// Mitsubishi GX Works2 project: PID_slave_test_fx3u_demo   PLC: FX3U/FX3UC

// global labels: Global1
VAR_GLOBAL
  Input_ManualMode AT M500 : BOOL;  (* Valg av Manuell "1" eller Auto "0" *)
  Input_OperationModus AT M501 : BOOL;  (* Valg av direkte "1" eller Revers "0" Regulering *)
  Input_IntegratorModus AT M502 : BOOL;  (* Valg av Integrator virkning på regulator *)
  Input_DerivatorModus AT M503 : BOOL;  (* Valg av Derivator virkning på regulator *)
  Input_SamplingsTime AT D200 : INT;  (* Samplingstid sendt til PID *)
  Output_PID AT D202 : REAL;  (* Utgangs signal sendt ut fra PID *)
  Input_Referance AT D204 : REAL;  (* Referanse verdi sendt til PID *)
  Input_Process AT D206 : REAL;  (* Prosess verdi Sendt til PID *)
  Input_ManualValue AT D208 : REAL;  (* Manuell verdi sendt til PID *)
  Input_NomValue AT D210 : REAL;  (* Nominelt pådrag *)
  Input_MaxPådrag AT D212 : REAL;  (* Max pådrag *)
  Input_MinPådrag AT D214 : REAL;  (* Min pådrag *)
  Input_Skalert_Samplingstid AT D216 : ARRAY [0..1] OF INT;  (* Samplingstid skalert til timer *)
  Input_KpValue AT D218 : REAL;  (* Valg av Kp verdi *)
  Input_TiValue AT D220 : REAL;  (* Valge av Ti verdi *)
  Input_TdValue AT D222 : REAL;  (* Valg av Td verdi *)
  Input_NValue AT D224 : REAL;  (* Valg av N verdi *)
  Input_TtValue AT D226 : REAL;  (* Valg av Tt verdi *)
  Input_FF_TtValue AT D228 : REAL;  (* Valg av Tt verdi til LeadLag blokk *)
  Input_FF_TnValue AT D230 : REAL;  (* Valg av Tn verdi til LeadLag blokk *)
  Input_FF_KLLValue AT D232 : REAL;  (* Valg av KLL verdi til LeadLag blokk *)
  Output_Leadlag AT D234 : REAL;  (* Utgangsignal sendt ut fra LeadLag blokk *)
  Output_Total AT D236 : REAL;  (* Totalt utgangsignal summert *)
  Input_ErrorValue AT D238 : REAL;  (* Beregnet avvik *)
  Input_AI_Raw AT D400 : INT;
  Output_AO_Raw AT D402 : INT;
  Storage_havardsinlillepikk AT D500 : INT;  (* Mellomlagrin av referanse verdi før omgjøring til flyttall *)
  anaDig AT D8260 : INT;
  digAna AT D8262 : INT;
  Storage_Filter_Output AT D502 : INT;  (* Utgangsverdi fra filter *)
  Tank_high AT M504 : BOOL;
  Tank_low AT M505 : BOOL;
  Tank_high_high AT M506 : BOOL;
  Tank_low_low AT M507 : BOOL;
  Tank_criticalHigh AT M508 : BOOL;
  Tank_criticalLow AT M509 : BOOL;
  Tank_normalHigh AT M510 : BOOL;
  Tank_normalLow AT M511 : BOOL;
  Acknowledge_normalHigh AT M512 : BOOL;
  Acknowledge_normalLow AT M513 : BOOL;
  Acknowledge_criticalHigh AT M514 : BOOL;
  Acknowledge_criticalLow AT M515 : BOOL;
  Pump AT Y012 : BOOL;
  Normal_ErrorSignal AT M516 : BOOL;
  Critical_ErrorSignal AT M517 : BOOL;
  Normal_ErrorCheck AT M518 : ARRAY [0..2] OF BOOL;
  Critical_ErrorCheck AT M519 : ARRAY [0..2] OF BOOL;
  Process_memory AT M520 : BOOL;
  Process AT M21 : BOOL;
  Power_failure AT M522 : BOOL;
  Acknowledge_powerFailure AT M523 : BOOL;
  Alarm_Lamp AT Y001 : BOOL;
  Communication_trouble AT X001 : BOOL;
  Communication_troubleRST AT Y002 : BOOL;
  Communication_troubleRSTCommand AT X021 : BOOL;
  Communication_rstFlag AT M1 : BOOL;
  Profibus_code AT D1000 : INT;
END_VAR

// task Task_01 (event TRUE, interval 0, priority 31): POU_01

PROGRAM POU_01
VAR
  My_PID_1 : My_PID;
  LeadLag_1 : LeadLag;
  Output_Adder_1 : Output_Adder;
  Filter_Midling_1 : Filter_Midling;
END_VAR
(* structured ladder/FBD written out as ST: instructions are called as NAME(EN, inputs, outputs); _pN, _eN, _tN stand for wires *)
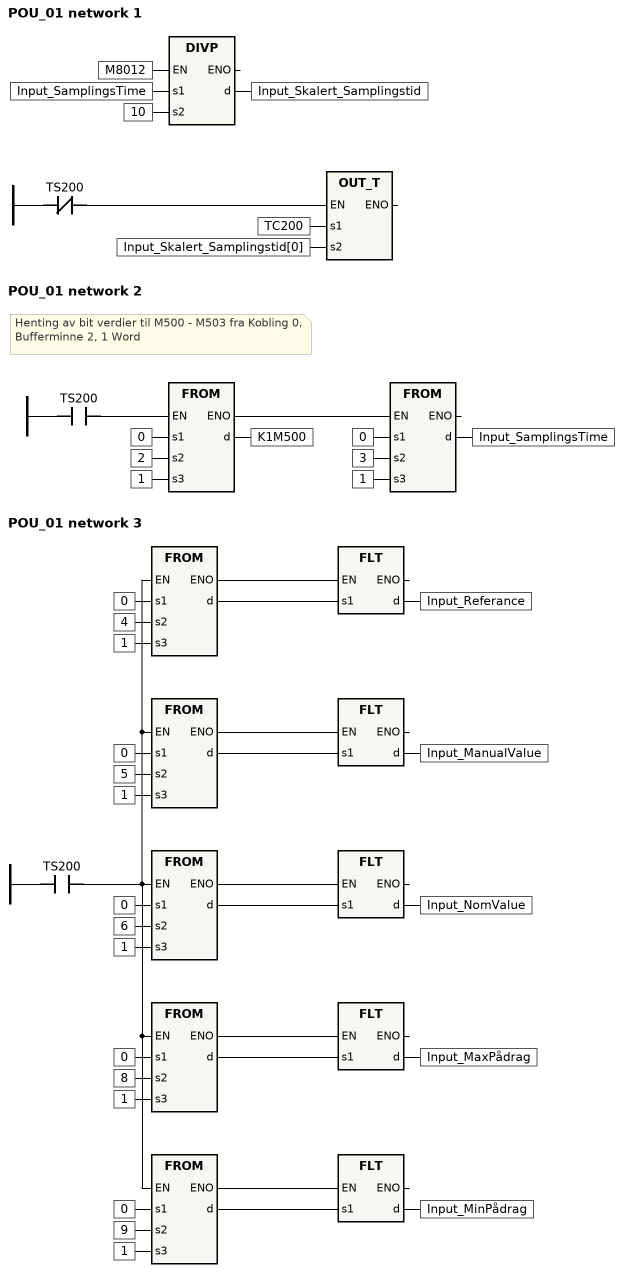
(* network 1 *)
DIVP(M8012, Input_SamplingsTime, 10, Input_Skalert_Samplingstid);
OUT_T(NOT TS200, TC200, Input_Skalert_Samplingstid[0]);
(* network 2 *)
(* Henting av bit verdier til M500 - M503 fra Kobling 0, Bufferminne 2, 1 Word *)
_e1 := FROM(TS200, 0, 2, 1, K1M500);
FROM(_e1, 0, 3, 1, Input_SamplingsTime);
(* network 3 *)
_e2 := FROM(TS200, 0, 4, 1, _t1);
FLT(_e2, _t1, Input_Referance);
_e4 := FROM(TS200, 0, 5, 1, _t3);
FLT(_e4, _t3, Input_ManualValue);
_e6 := FROM(TS200, 0, 6, 1, _t5);
FLT(_e6, _t5, Input_NomValue);
_e8 := FROM(TS200, 0, 8, 1, _t7);
FLT(_e8, _t7, Input_MaxPådrag);
_e10 := FROM(TS200, 0, 9, 1, _t9);
FLT(_e10, _t9, Input_MinPådrag);
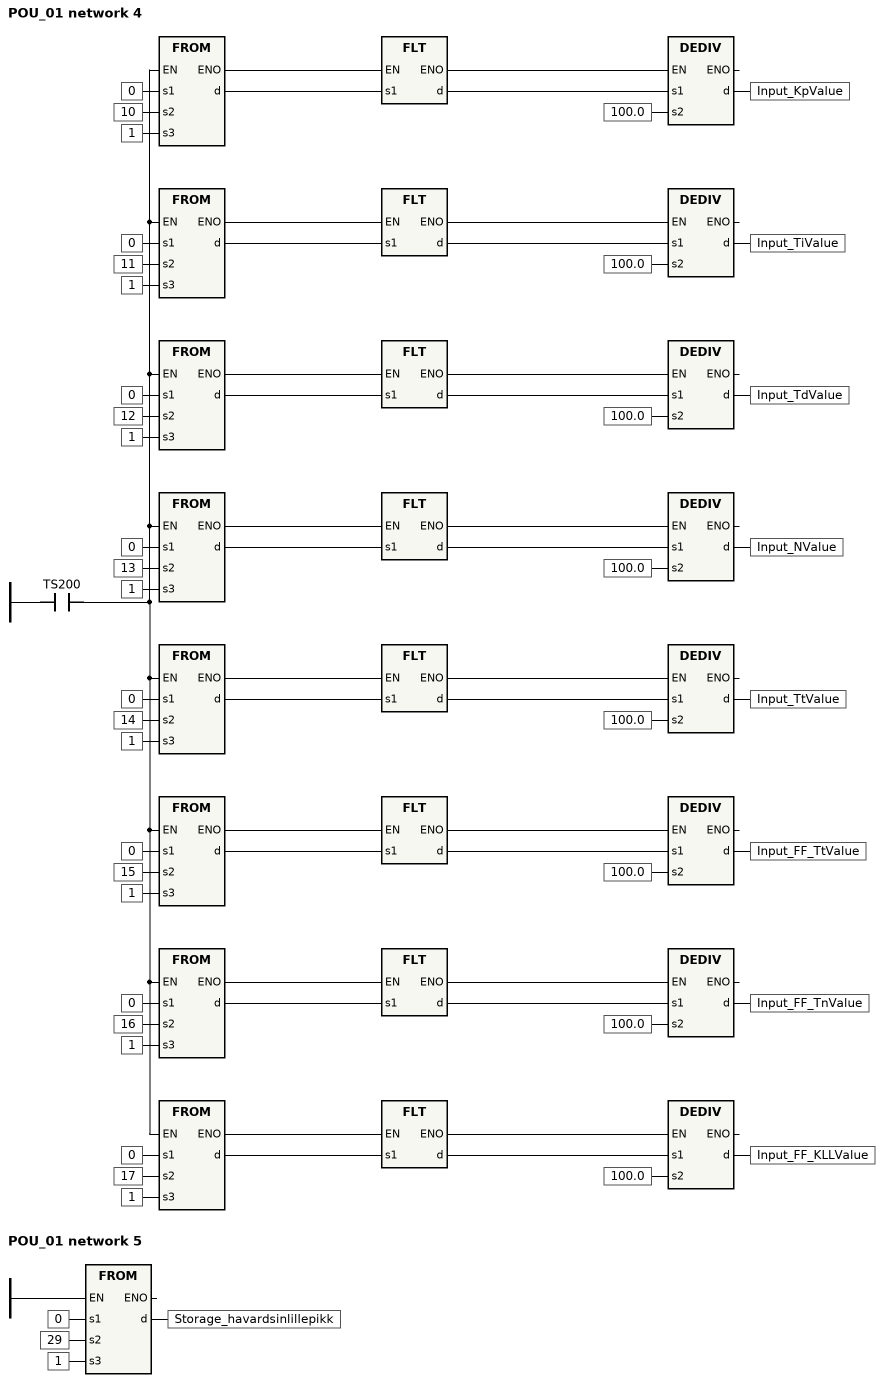
(* network 4 *)
_e2 := FROM(TS200, 0, 10, 1, _t1);
_e4 := FLT(_e2, _t1, _t3);
DEDIV(_e4, _t3, 100.0, Input_KpValue);
_e6 := FROM(TS200, 0, 11, 1, _t5);
_e8 := FLT(_e6, _t5, _t7);
DEDIV(_e8, _t7, 100.0, Input_TiValue);
_e10 := FROM(TS200, 0, 12, 1, _t9);
_e12 := FLT(_e10, _t9, _t11);
DEDIV(_e12, _t11, 100.0, Input_TdValue);
_e14 := FROM(TS200, 0, 13, 1, _t13);
_e16 := FLT(_e14, _t13, _t15);
DEDIV(_e16, _t15, 100.0, Input_NValue);
_e18 := FROM(TS200, 0, 14, 1, _t17);
_e20 := FLT(_e18, _t17, _t19);
DEDIV(_e20, _t19, 100.0, Input_TtValue);
_e22 := FROM(TS200, 0, 15, 1, _t21);
_e24 := FLT(_e22, _t21, _t23);
DEDIV(_e24, _t23, 100.0, Input_FF_TtValue);
_e26 := FROM(TS200, 0, 16, 1, _t25);
_e28 := FLT(_e26, _t25, _t27);
DEDIV(_e28, _t27, 100.0, Input_FF_TnValue);
_e30 := FROM(TS200, 0, 17, 1, _t29);
_e32 := FLT(_e30, _t29, _t31);
DEDIV(_e32, _t31, 100.0, Input_FF_KLLValue);
(* network 5 *)
FROM(TRUE, 0, 29, 1, Storage_havardsinlillepikk);
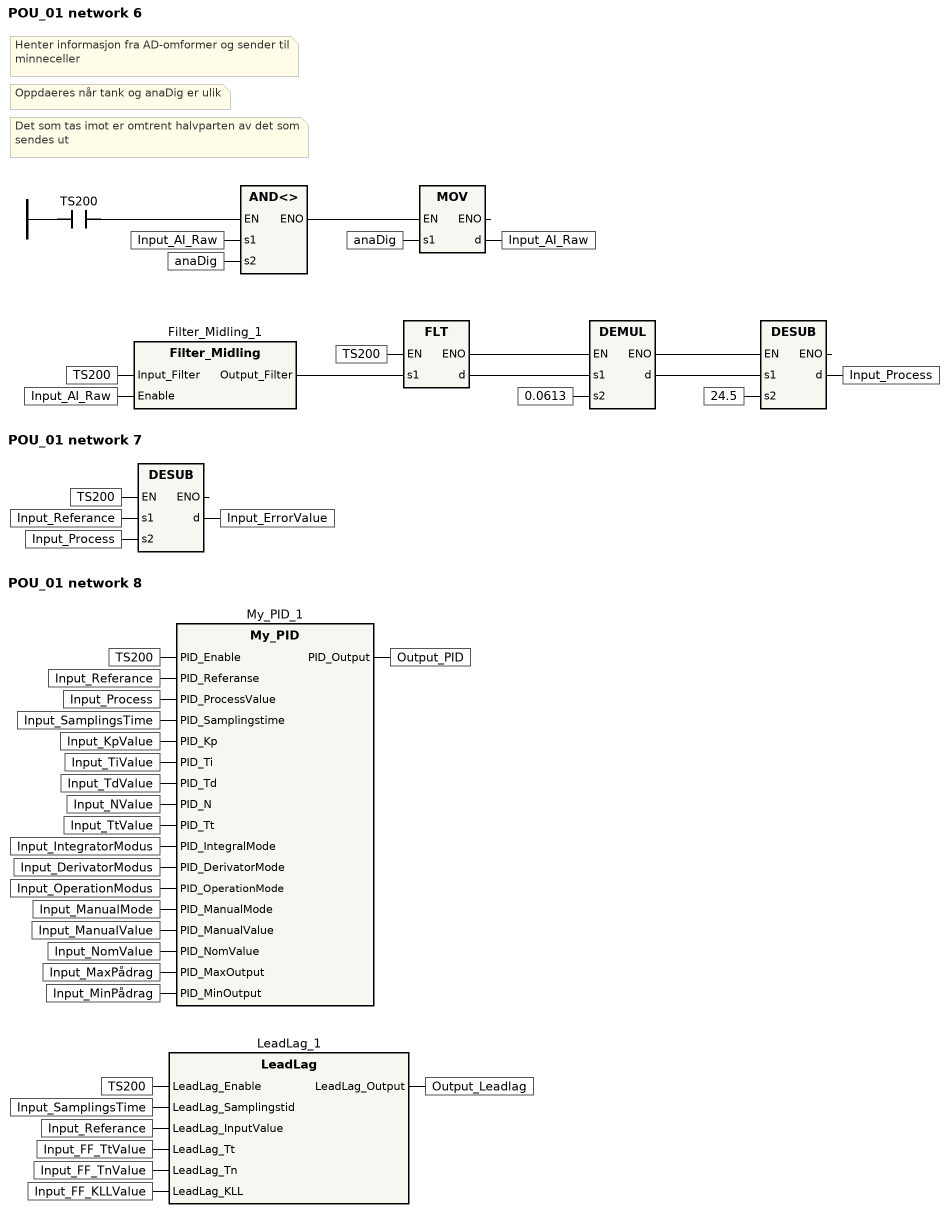
(* network 6 *)
(* Henter informasjon fra AD-omformer og sender til minneceller *)
(* Oppdaeres når tank og anaDig er ulik *)
(* Det som tas imot er omtrent halvparten av det som sendes ut *)
_e1 := AND<>(TS200, Input_AI_Raw, anaDig);
MOV(_e1, anaDig, Input_AI_Raw);
Filter_Midling_1(Input_Filter := TS200, Enable := Input_AI_Raw);
_e3 := FLT(TS200, Filter_Midling_1.Output_Filter, _t2);
_e5 := DEMUL(_e3, _t2, 0.0613, _t4);
DESUB(_e5, _t4, 24.5, Input_Process);
(* network 7 *)
DESUB(TS200, Input_Referance, Input_Process, Input_ErrorValue);
(* network 8 *)
My_PID_1(PID_Enable := TS200, PID_Referanse := Input_Referance, PID_ProcessValue := Input_Process, PID_Samplingstime := Input_SamplingsTime, PID_Kp := Input_KpValue, PID_Ti := Input_TiValue, PID_Td := Input_TdValue, PID_N := Input_NValue, PID_Tt := Input_TtValue, PID_IntegralMode := Input_IntegratorModus, PID_DerivatorMode := Input_DerivatorModus, PID_OperationMode := Input_OperationModus, PID_ManualMode := Input_ManualMode, PID_ManualValue := Input_ManualValue, PID_NomValue := Input_NomValue, PID_MaxOutput := Input_MaxPådrag, PID_MinOutput := Input_MinPådrag, PID_Output => Output_PID);
LeadLag_1(LeadLag_Enable := TS200, LeadLag_Samplingstid := Input_SamplingsTime, LeadLag_InputValue := Input_Referance, LeadLag_Tt := Input_FF_TtValue, LeadLag_Tn := Input_FF_TnValue, LeadLag_KLL := Input_FF_KLLValue, LeadLag_Output => Output_Leadlag);
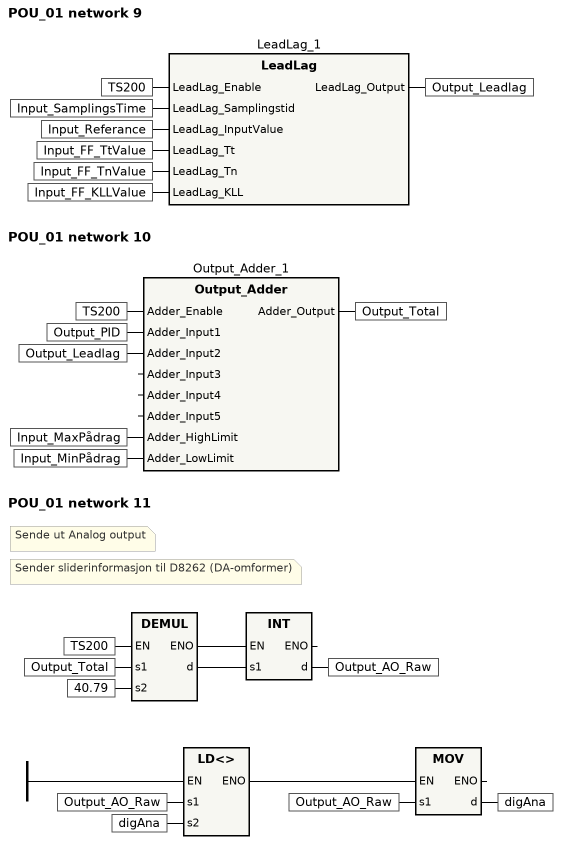
(* network 9 *)
LeadLag_1(LeadLag_Enable := TS200, LeadLag_Samplingstid := Input_SamplingsTime, LeadLag_InputValue := Input_Referance, LeadLag_Tt := Input_FF_TtValue, LeadLag_Tn := Input_FF_TnValue, LeadLag_KLL := Input_FF_KLLValue, LeadLag_Output => Output_Leadlag);
(* network 10 *)
Output_Adder_1(Adder_Enable := TS200, Adder_Input1 := Output_PID, Adder_Input2 := Output_Leadlag, Adder_HighLimit := Input_MaxPådrag, Adder_LowLimit := Input_MinPådrag, Adder_Output => Output_Total);
(* network 11 *)
(* Sende ut Analog output *)
(* Sender sliderinformasjon til D8262 (DA-omformer) *)
_e2 := DEMUL(TS200, Output_Total, 40.79, _t1);
INT(_e2, _t1, Output_AO_Raw);
_e3 := LD<>(TRUE, Output_AO_Raw, digAna);
MOV(_e3, Output_AO_Raw, digAna);
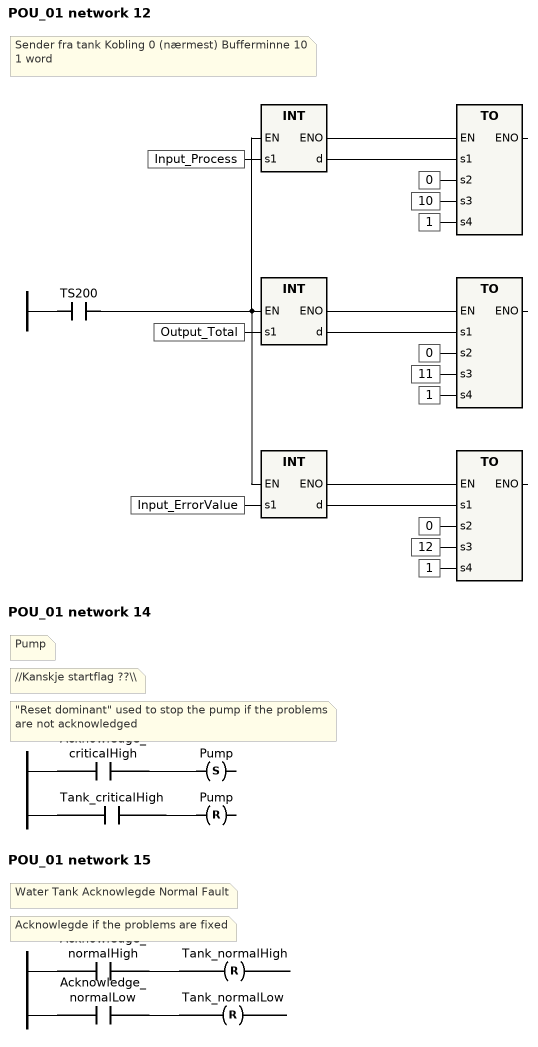
(* network 12 *)
(* Sender fra tank Kobling 0 (nærmest) Bufferminne 10           1 word *)
_e2 := INT(TS200, Input_Process, _t1);
TO(_e2, _t1, 0, 10, 1);
_e4 := INT(TS200, Output_Total, _t3);
TO(_e4, _t3, 0, 11, 1);
_e6 := INT(TS200, Input_ErrorValue, _t5);
TO(_e6, _t5, 0, 12, 1);
(* network 14 *)
(* Pump *)
(* //Kanskje startflag ??\\ *)
(* "Reset dominant" used to stop the pump if the problems are not acknowledged *)
SET(Acknowledge_criticalHigh, Pump);
RST(Tank_criticalHigh, Pump);
(* network 15 *)
(* Water Tank Acknowlegde Normal Fault *)
(* Acknowlegde if the problems are fixed *)
RST(Acknowledge_normalHigh, Tank_normalHigh);
RST(Acknowledge_normalLow, Tank_normalLow);
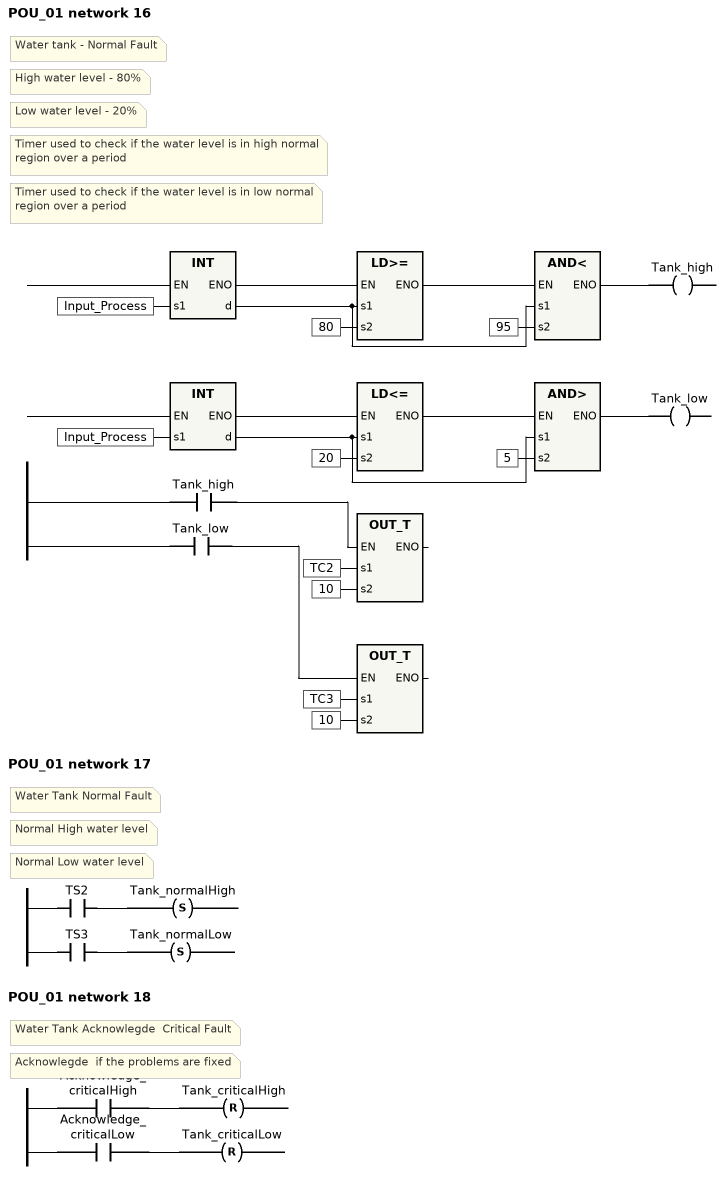
(* network 16 *)
(* Water tank - Normal Fault *)
(* High water level - 80% *)
(* Low water level - 20% *)
(* Timer used to check if the water level is in high normal region over a period *)
(* Timer used to check if the water level is in low normal region over a period *)
_e2 := INT(TRUE, Input_Process, _t1);
_e3 := LD>=(_e2, _t1, 80);
_e4 := AND<(_e3, _t1, 95);
Tank_high := _e4;
_e6 := INT(TRUE, Input_Process, _t5);
_e7 := LD<=(_e6, _t5, 20);
_e8 := AND>(_e7, _t5, 5);
Tank_low := _e8;
OUT_T(Tank_high, TC2, 10);
OUT_T(Tank_low, TC3, 10);
(* network 17 *)
(* Water Tank Normal Fault *)
(* Normal High water level *)
(* Normal Low water level *)
SET(TS2, Tank_normalHigh);
SET(TS3, Tank_normalLow);
(* network 18 *)
(* Water Tank Acknowlegde  Critical Fault *)
(* Acknowlegde  if the problems are fixed *)
RST(Acknowledge_criticalHigh, Tank_criticalHigh);
RST(Acknowledge_criticalLow, Tank_criticalLow);
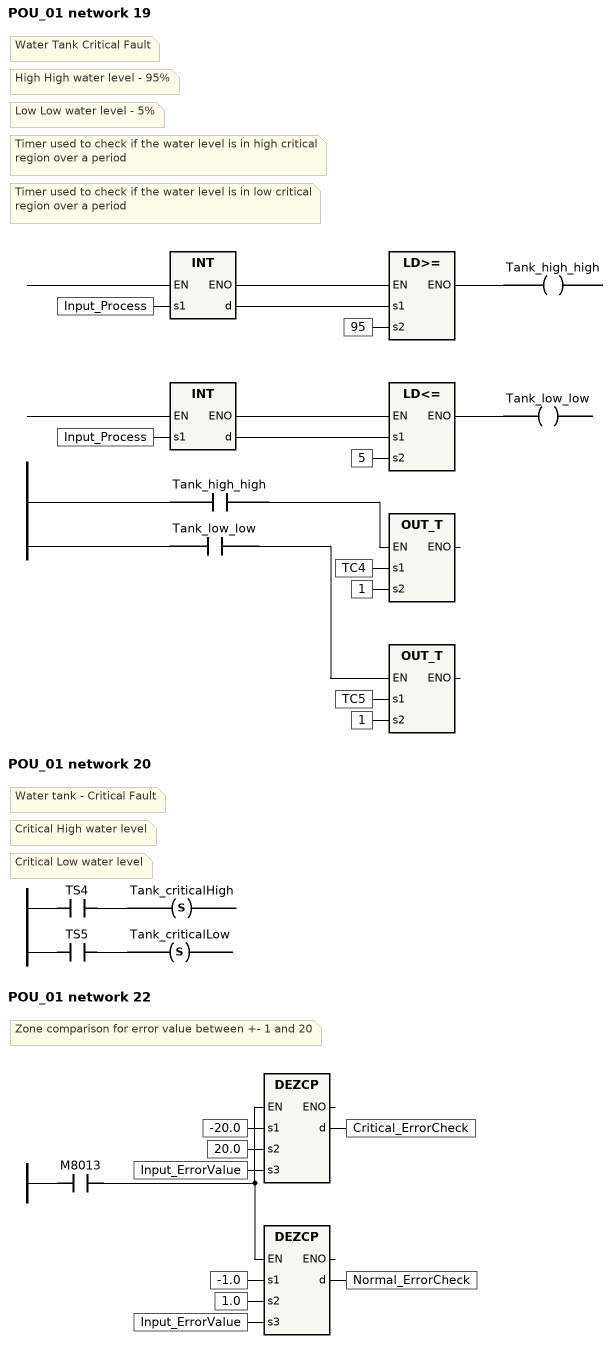
(* network 19 *)
(* Water Tank Critical Fault *)
(* High High water level - 95% *)
(* Low Low water level - 5% *)
(* Timer used to check if the water level is in high critical region over a period *)
(* Timer used to check if the water level is in low critical region over a period *)
_e2 := INT(TRUE, Input_Process, _t1);
_e3 := LD>=(_e2, _t1, 95);
Tank_high_high := _e3;
_e5 := INT(TRUE, Input_Process, _t4);
_e6 := LD<=(_e5, _t4, 5);
Tank_low_low := _e6;
OUT_T(Tank_high_high, TC4, 1);
OUT_T(Tank_low_low, TC5, 1);
(* network 20 *)
(* Water tank - Critical Fault *)
(* Critical High water level *)
(* Critical Low water level *)
SET(TS4, Tank_criticalHigh);
SET(TS5, Tank_criticalLow);
(* network 22 *)
(* Zone comparison for error value between +- 1 and 20 *)
DEZCP(M8013, -20.0, 20.0, Input_ErrorValue, Critical_ErrorCheck);
DEZCP(M8013, -1.0, 1.0, Input_ErrorValue, Normal_ErrorCheck);
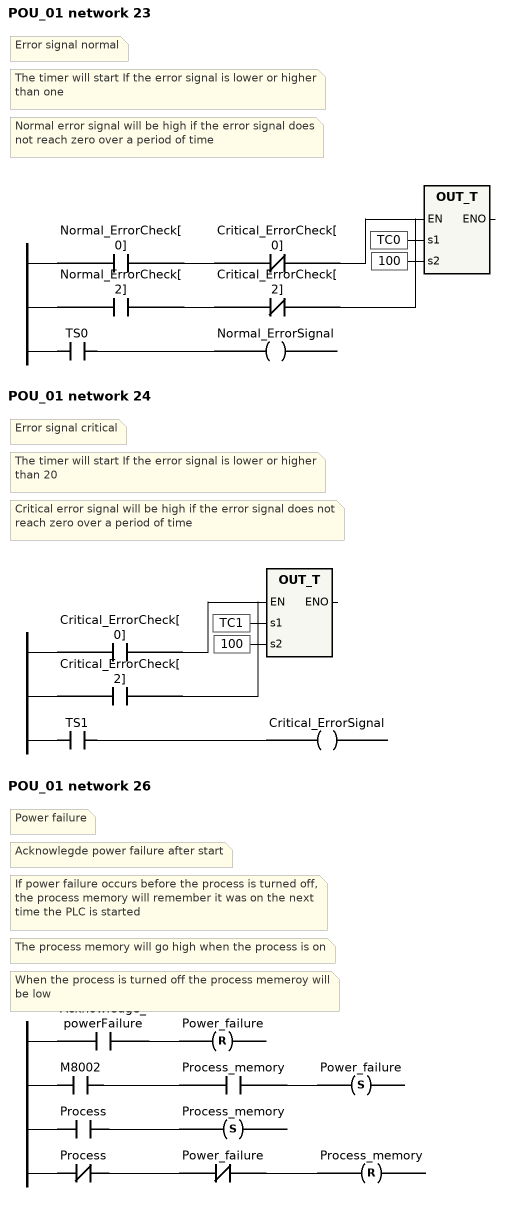
(* network 23 *)
(* Error signal normal *)
(* The timer will start If the error signal is lower or higher than one *)
(* Normal error signal will be high if the error signal does not reach zero over a period of time *)
OUT_T((Normal_ErrorCheck[0] AND NOT Critical_ErrorCheck[0]) OR (Normal_ErrorCheck[2] AND NOT Critical_ErrorCheck[2]), TC0, 100);
Normal_ErrorSignal := TS0;
(* network 24 *)
(* Error signal critical *)
(* The timer will start If the error signal is lower or higher than 20 *)
(* Critical error signal will be high if the error signal does not reach zero over a period of time *)
OUT_T(Critical_ErrorCheck[0] OR Critical_ErrorCheck[2], TC1, 100);
Critical_ErrorSignal := TS1;
(* network 26 *)
(* Power failure *)
(* Acknowlegde power failure after start *)
(* If power failure occurs before the process is turned off, the process memory will remember it was on the next time the PLC is started *)
(* The process memory will go high when the process is on *)
(* When the process is turned off the process memeroy will be low *)
RST(Acknowledge_powerFailure, Power_failure);
SET(M8002 AND Process_memory, Power_failure);
SET(Process, Process_memory);
RST(NOT Process AND NOT Power_failure, Process_memory);
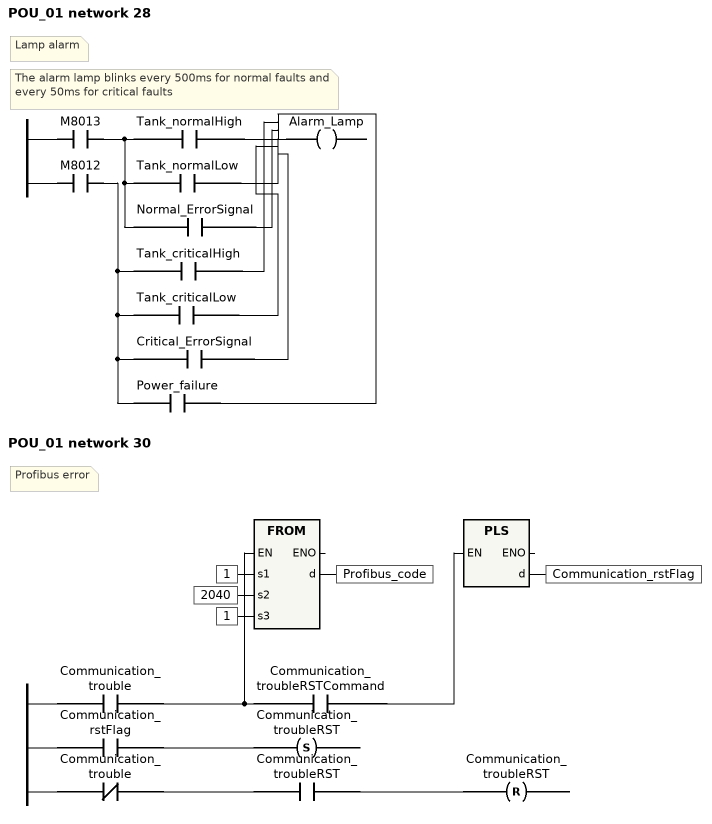
(* network 28 *)
(* Lamp alarm *)
(* The alarm lamp blinks every 500ms for normal faults and every 50ms for critical faults *)
Alarm_Lamp := (M8013 AND Tank_normalHigh) OR (M8013 AND Tank_normalLow) OR (M8013 AND Normal_ErrorSignal) OR (M8012 AND Tank_criticalHigh) OR (M8012 AND Tank_criticalLow) OR (M8012 AND Critical_ErrorSignal) OR (M8012 AND Power_failure);
(* network 30 *)
(* Profibus error *)
FROM(Communication_trouble, 1, 2040, 1, Profibus_code);
PLS(Communication_trouble AND Communication_troubleRSTCommand, Communication_rstFlag);
SET(Communication_rstFlag, Communication_troubleRST);
RST(NOT Communication_trouble AND Communication_troubleRST, Communication_troubleRST);
END_PROGRAM

FUNCTION_BLOCK My_PID
VAR_INPUT
  PID_Enable : BOOL;  (* Samplings enable *)
  PID_Referanse : REAL;  (* Referanseverdi PID blokk *)
  PID_ProcessValue : REAL;  (* Prosessverdi PID blokk *)
  PID_Samplingstime : INT;  (* Samplingstid PID blokk (ms) *)
  PID_Kp : REAL;  (* KP PID blokk *)
  PID_Ti : REAL;  (* Ti PID blokk *)
  PID_Td : REAL;  (* Td PID blokk *)
  PID_N : REAL;  (* Filter konstant for Tf *)
  PID_Tt : REAL;  (* Tracking konstant for PID tracking inngang *)
  PID_IntegralMode : BOOL;  (* Integrator for PID blokk *)
  PID_DerivatorMode : BOOL;  (* Derivator for PID blokk *)
  PID_OperationMode : BOOL;  (* Direkte kobling "1", reversert "0" *)
  PID_ManualMode : BOOL;  (* Auto "0" , Manuell pådrag "1" *)
  PID_ManualValue : REAL;  (* Manuelt pådrag verdi *)
  PID_NomValue : REAL;  (* Nominelt pådrags verdi *)
  PID_MaxOutput : REAL;  (* Max pådrags verdi *)
  PID_MinOutput : REAL;  (* Min pådrags verdi *)
END_VAR
VAR_OUTPUT
  PID_Output : REAL;  (* Utgangsverdi fra PID-reg *)
END_VAR
VAR
  PID_Alpha : REAL;  (* Beregnet alpha verdi *)
  PID_Beta : REAL;  (* Beregnet betaverdi *)
  PID_Gamma : REAL;  (* Beregnet gammaverdi *)
  PID_ErrorValue_F : ARRAY [0..1] OF REAL;  (* Beregnet error verdi (Denne og forrige verdi) *)
  PID_PGain : ARRAY [0..1] OF REAL;  (* Beregnet P forsterkning (Denne og forrige verdi) *)
  PID_IGain : ARRAY [0..1] OF REAL;  (* Beregnet I forsterkning (Denne og forrige verdi) *)
  PID_DGain : ARRAY [0..1] OF REAL;  (* Beregnet D forsterkning (Denne og forrige verdi) *)
  PID_Gain_Total : REAL;  (* Beregnet sum av total pådrag (Ubegrenset verdi) *)
  PID_Gain_Tracking : REAL;  (* Beregnet sum av tracking pådrag (Begrenset verdi) *)
  PID_ProcessValue_F : ARRAY [0..1] OF REAL;  (* Prosess verdi i PID blokk (denne og forrige verdi) *)
  PID_Scaled_Samplingstime : REAL;  (* Skalert samplingstid i sekunder *)
  PID_Calc_Sampling : REAL;  (* Mellomregning av samplingstid *)
END_VAR
(*Omgjøring av samplingstid fra ms til s*)
FLT(TRUE , PID_Samplingstime, PID_Calc_Sampling);
PID_Scaled_Samplingstime := PID_Calc_Sampling/1000.0;



(*Systemet vil gå inn i koden hvert samplingstid som er satt*)

IF PID_Enable THEN	
	
	
	(*Regning av konstanter alpha, beta, gamma og lagring av prosessverdi til et array*)
	PID_Alpha := PID_Scaled_Samplingstime/PID_Ti;
	PID_Beta := PID_Td/(PID_Td + (PID_Scaled_Samplingstime*pid_n));
	PID_Gamma:= PID_Scaled_Samplingstime/PID_Tt;
	PID_ProcessValue_F[0] := PID_ProcessValue;

	
	(*Regning av avvik mtp om det er direkte eller revers regulering*)
	IF PID_OperationMode THEN
		PID_ErrorValue_F[0] := PID_ProcessValue_F[0] - PID_Referanse;
	ELSE
		PID_ErrorValue_F[0] := PID_Referanse - PID_ProcessValue_F[0];
	END_IF;
	

	(*Beregning av pådragsbidrag fra P-del*)
	PID_PGain[0] := PID_Kp*PID_ErrorValue_F[0];
	
	(*Ser om integrator er aktivert og beregner pådragsbidrag fra I-del med tracking inngang*)
	IF PID_IntegralMode THEN
		PID_IGain[0] := PID_IGain[1] + PID_Kp*PID_Alpha*PID_ErrorValue_F[0]+PID_Gamma*(PID_Gain_Tracking-PID_Gain_Total);
	ELSE
		PID_IGain[0] := 0.0;
	END_IF;
	
	(*Ser om Derivator er aktivert og beregner pådragsbidrag fra D-del*)
	IF PID_DerivatorMode THEN
		PID_DGain[0] := (PID_Beta*PID_DGain[1]) - ((PID_Kp*PID_Td/PID_Scaled_Samplingstime)*(1.0-PID_Beta)*(PID_ProcessValue_F[0]-PID_ProcessValue_F[1]));
	ELSE 
		PID_DGain[0] := 0.0;
	END_IF;
	
	(*Summerer sammen pådragsbidrag fra alle delene*)
	PID_Gain_Total := PID_PGain[0] + PID_IGain[0] + PID_DGain[0] + PID_NomValue;
	
	(*Oppdatering av verdier*)
	PID_ErrorValue_F[1] := PID_ErrorValue_F[0];
	PID_ProcessValue_F[1] := PID_ProcessValue_F[0];
	PID_PGain[1] := PID_PGain[0];
	PID_IGain[1] := PID_IGain[0];
	PID_DGain[1] := PID_DGain[0];
	
	(*Ser om regulatoren skal gå i auto eller manuell modus*)
	IF PID_ManualMode THEN 
		PID_Gain_Tracking := PID_ManualValue;
	ELSE 
		PID_Gain_Tracking := PID_Gain_Total;
	END_IF;
	
	(*Kontrollerer at pådragsbidrag er innenfor min og max verdier*)
	IF PID_Gain_Tracking > PID_maxoutput THEN
		PID_Gain_Tracking:= PID_MaxOutput ;
	ELSIF PID_Gain_Tracking< PID_MinOutput THEN 
		PID_Gain_Tracking:= PID_MinOutput;
	ELSE
		PID_Gain_Tracking:= PID_Gain_Tracking;
	END_IF;
	
	(*Utgang fra PID regulator*)
	PID_Output := PID_Gain_Tracking;
ELSE 
;
END_IF;
END_FUNCTION_BLOCK

FUNCTION_BLOCK LeadLag
VAR_INPUT
  LeadLag_Enable : BOOL;  (* Enable for hvert samplingstid *)
  LeadLag_Samplingstid : INT;  (* Samplingstid Lead Lag blokk *)
  LeadLag_InputValue : REAL;  (* Inngangsverdi inn til LeadLag blokk *)
  LeadLag_Tt : REAL;  (* Tt konstant for Lead Lag blokk *)
  LeadLag_Tn : REAL;  (* Tn konstant for Lead Lag blokk *)
  LeadLag_KLL : REAL;  (* KLL konstant for Lead Lag blokk *)
END_VAR
VAR_OUTPUT
  LeadLag_Output : REAL;  (* Utgangsverdu ut fra LeadLag blokk *)
END_VAR
VAR
  LeadLag_Mellomregning_Sampl : REAL;  (* Mellom regning for samplingstid *)
  LeadLag_Skalert_Samplingstid : REAL;  (* Skalert samplingstid i sekunder *)
  LeadLag_InputValue_F : ARRAY [0..1] OF REAL;  (* Input verdi denne og forrige *)
  LeadLag_Output_F : ARRAY [0..1] OF REAL;  (* Utgangspådrag  (denne og forrige) *)
END_VAR
(*Omgjøring av samplingstid fra ms til s*)
FLT(TRUE , leadlag_Samplingstid, leadLag_Mellomregning_Sampl);
LeadLag_Skalert_Samplingstid := leadlag_Mellomregning_Sampl/1000.0;

IF LeadLag_Enable THEN
	LeadLag_InputValue_F[0] := LeadLag_InputValue;
	
	LeadLag_Output_F[0] := (LeadLag_KLL*((LeadLag_Tt+LeadLag_Skalert_Samplingstid)*LeadLag_InputValue_F[0]-LeadLag_Tt*LeadLag_InputValue_F[1])+LeadLag_Tn*LeadLag_Output_F[1])/(LeadLag_Tn+LeadLag_Skalert_Samplingstid);
	
	LeadLag_Output_F[1] := LeadLag_Output_F[0];
	LeadLag_InputValue_F[1] := LeadLag_InputValue_F[0];
	
	LeadLag_Output := LeadLag_Output_F[0];
ELSE

;
END_IF;


;
END_FUNCTION_BLOCK

FUNCTION_BLOCK Output_Adder
VAR_INPUT
  Adder_Enable : BOOL;
  Adder_Input1 : REAL;  (* Input value 1 *)
  Adder_Input2 : REAL;  (* Input value 2 *)
  Adder_Input3 : REAL;  (* Input value 3 *)
  Adder_Input4 : REAL;  (* Input value 4 *)
  Adder_Input5 : REAL;  (* Input value 5 *)
  Adder_HighLimit : REAL;  (* Maximum output *)
  Adder_LowLimit : REAL;  (* Minimum output *)
END_VAR
VAR_OUTPUT
  Adder_Output : REAL;  (* Total output from adder *)
END_VAR
VAR
  Adder_Sum : REAL;  (* Sum av inputs *)
END_VAR
IF Adder_Enable THEN
	Adder_Sum := Adder_Input1+Adder_Input2+Adder_Input3+Adder_Input4+Adder_Input5;
	
	IF Adder_Sum > Adder_HighLimit THEN
		Adder_Output := Adder_HighLimit;
	ELSIF Adder_Sum < Adder_LowLimit THEN
		Adder_Output := Adder_LowLimit;
	ELSE
		Adder_Output := Adder_Sum;
	END_IF;
END_IF;
;
END_FUNCTION_BLOCK

FUNCTION_BLOCK Filter_Midling
VAR_INPUT
  Input_Filter : INT;  (* Inngangs verdi til filter *)
END_VAR
VAR_OUTPUT
  Output_Filter : INT;  (* Utgangsverdi til filter *)
END_VAR
VAR
  Input_Array : ARRAY [0..2] OF INT;  (* Array av inngangsverdier *)
END_VAR
VAR_INPUT
  Enable : BOOL;  (* Enabler *)
END_VAR
Input_Array[0] := Input_Filter;

Output_Filter:=  (Input_Array[0] + Input_Array[1] + Input_Array[2])/3;

Input_Array[2]:= Input_Array[1];
Input_Array[1] := Input_Array[0];


;
END_FUNCTION_BLOCK
